TYPE ST_PNOZRawOut :
STRUCT
    abyOutput: ARRAY[1..GVL_SafetyIO.cPNOZ_RXPDO_BYTES] OF BYTE; //Output Byte 00..18 (0-144 bits)
END_STRUCT
END_TYPE

(* stored: Version 1.1.0.1
   DUT ST_PNOZRawOut: Id {f721d84d-ba9b-4caa-9515-51e70651d496} *)
